Omron Sysmac Studio project Auto Connect Project (Sysmac Studio 1.48.0.8, StandardProject)

# Controller new_Controller_0: NX102-1020 version 1.35
Units and slaves: Unit 1 : NX-CIF101 (N1); Unit 2 : NX-ID5142-1 (N2); Unit 3 : NX-OD5121-1 (N3)
Task PrimaryTask (priority 4, period or condition 2000): Program0

VAR_GLOBAL RETAIN
    data1 : INT;
END_VAR
VAR_GLOBAL
    data2 : INT;
    data3 : INT;
    data4 : INT;
    data5 : INT;
    dataA_1 : STRING[256];
    dataA_2 : STRING[256];
    dataA_3 : STRING[256];
    dataA_4 : STRING[256];
    dataA_5 : STRING[256];
    dataB_1 : REAL;
    dataB_2 : REAL;
    dataB_3 : REAL;
    dataB_4 : REAL;
    dataB_5 : REAL;
    senser1 : BOOL;
    pump1 : BOOL;
    pb_start : BOOL;
END_VAR

PROGRAM Program0
VAR
    start_1 : BOOL;
    stop_1 : BOOL;
    lam_1 : BOOL;
    lamp_1 : BOOL;
    sw_1 : BOOL;
    sw2 : BOOL;
    sw_2 : BOOL;
    lamp_2 : BOOL;
    sw3 : BOOL;
    sw4 : BOOL;
    lamp_3 : BOOL;
    sw5 : BOOL;
    lamp_4 : BOOL;
    sw_6 : BOOL;
    lamp_5 : BOOL;
    sw7 : BOOL;
    test_a : RS;
    sw_test_a : BOOL;
    lamp_6 : BOOL;
    sw_9 : BOOL;
    sww : BOOL;
    sw_8 : BOOL;
    test_b : BOOL;
    lamp_7 : BOOL;
    test_a_q1 : BOOL;
    sw_10 : BOOL;
    lamp_8 : BOOL;
    sw_11 : BOOL;
    test_b_1 : SR;
    t_on : BOOL;
    t_a1 : TON;
    pv1 : TIME;
    lamp_9 : BOOL;
    t_b1 : TOF;
    sw12 : BOOL;
    pv2 : TIME;
    lamp_10 : BOOL;
    sw13 : BOOL;
    t_c1 : TP;
    pv3 : TIME;
    lamp_11 : BOOL;
    sw14 : BOOL;
    t_d1 : AccumulationTimer;
    sw15 : BOOL;
    pv4 : TIME;
    lamp_12 : BOOL;
    C_A_D_C : CTU;
    box2 : BOOL;
    box1 : BOOL;
    pd_reset_1 : BOOL;
    cv_1 : INT;
    lamp_13 : BOOL;
    sw16 : BOOL;
    sw_17 : BOOL;
    sw_18 : BOOL;
    lamp_test : BOOL;
    sw_19 : BOOL;
    lamp_14 : BOOL;
    B1 : BOOL;
    B2 : BOOL;
    B3 : BOOL;
    B4 : BOOL;
    B5 : BOOL;
    B6 : BOOL;
    B7 : BOOL;
    lamp_15 : BOOL;
    p : BOOL;
END_VAR
VAR_EXTERNAL
    data1 : INT;
    data2 : INT;
    dataA_1 : STRING[256];
    dataA_2 : STRING[256];
    data3 : INT;
    data4 : INT;
    dataB_1 : REAL;
    dataB_2 : REAL;
    senser1 : BOOL;
    pump1 : BOOL;
END_VAR
VAR
    _t1 : BOOL;
    _e2 : F_TRIG;
    _e3 : R_TRIG;
    _e4 : R_TRIG;
END_VAR

(* Section Section0: ladder, written here as Structured Text *)

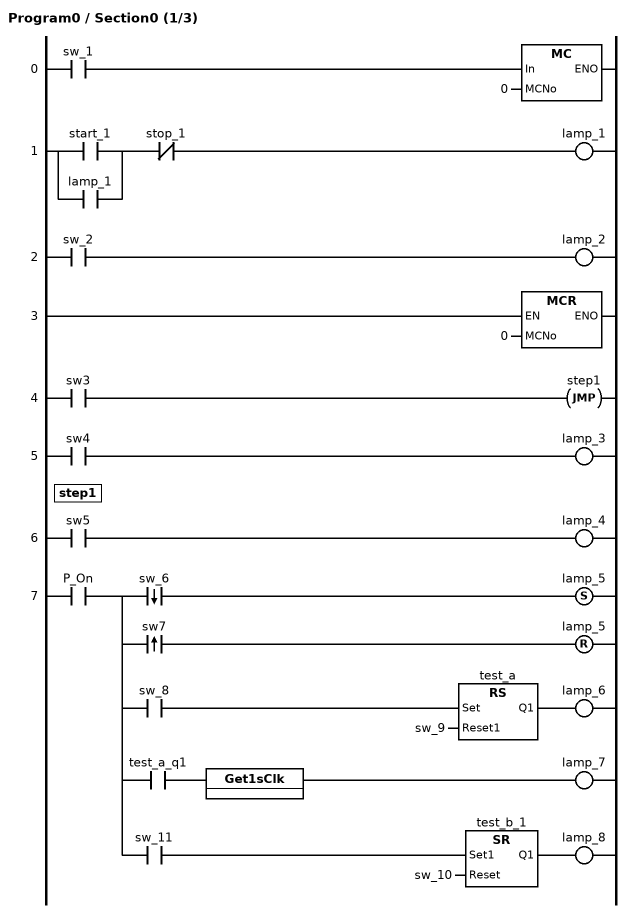
(* Rung 0 *)
MC(In := sw_1, MCNo := 0, ENO => _t1);
(* Rung 1 *)
lamp_1 := (start_1 OR lamp_1) AND NOT stop_1;
(* Rung 2 *)
lamp_2 := sw_2;
(* Rung 3 *)
MCR(MCNo := 0);
(* Rung 4 *)
IF sw3 THEN JMP step1; END_IF;
(* Rung 5 *)
lamp_3 := sw4;
(* Rung 6 *)
step1:
lamp_4 := sw5;
(* Rung 7 *)
_e2(CLK := sw_6);
IF P_On AND _e2.Q THEN lamp_5 := TRUE; END_IF;
_e3(CLK := sw7);
IF P_On AND _e3.Q THEN lamp_5 := FALSE; END_IF;
test_a(Set := P_On AND sw_8, Reset1 := sw_9);
lamp_6 := test_a.Q1;
lamp_7 := P_On AND test_a_q1 AND Get1sClk();
test_b_1(Set1 := P_On AND sw_11, Reset := sw_10);
lamp_8 := test_b_1.Q1;

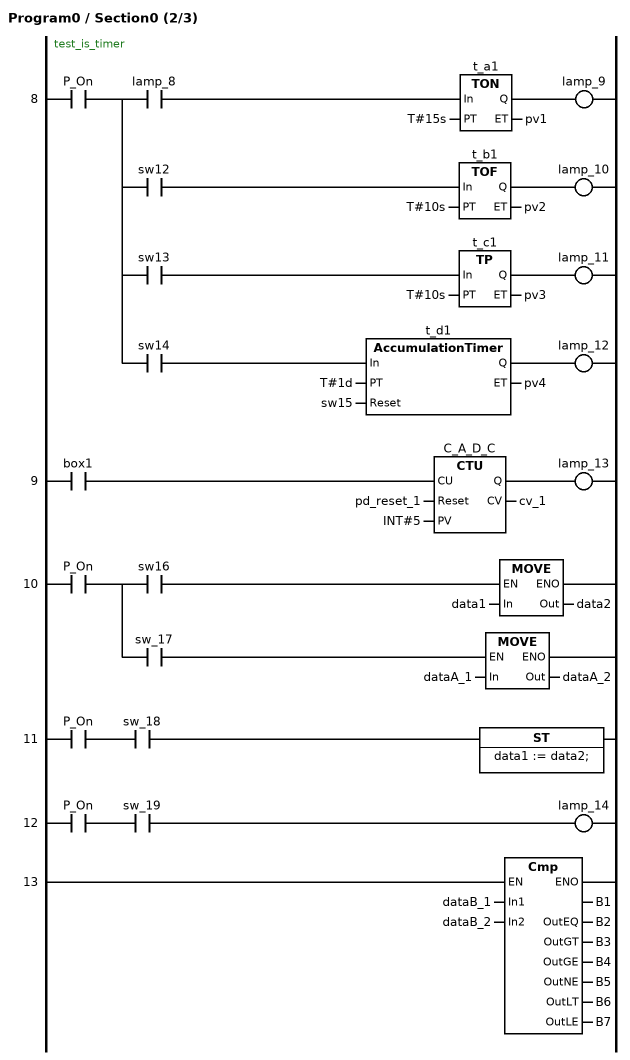
(* Rung 8: test_is_timer *)
t_a1(In := P_On AND lamp_8, PT := T#15s, ET => pv1);
lamp_9 := t_a1.Q;
t_b1(In := P_On AND sw12, PT := T#10s, ET => pv2);
lamp_10 := t_b1.Q;
t_c1(In := P_On AND sw13, PT := T#10s, ET => pv3);
lamp_11 := t_c1.Q;
t_d1(In := P_On AND sw14, PT := T#1d, Reset := sw15, ET => pv4);
lamp_12 := t_d1.Q;
(* Rung 9 *)
_e4(CLK := box1);
C_A_D_C(CU := _e4.Q, Reset := pd_reset_1, PV := INT#5, CV => cv_1);
lamp_13 := C_A_D_C.Q;
(* Rung 10 *)
IF P_On AND sw16 THEN data2 := data1; END_IF;
IF P_On AND sw_17 THEN dataA_2 := dataA_1; END_IF;
(* Rung 11 *)
IF P_On AND sw_18 THEN
    data1 := data2;
END_IF;
(* Rung 12 *)
lamp_14 := P_On AND sw_19;
(* Rung 13 *)
B1 := Cmp(In1 := dataB_1, In2 := dataB_2, OutEQ => B2, OutGT => B3, OutGE => B4, OutNE => B5, OutLT => B6, OutLE => B7);

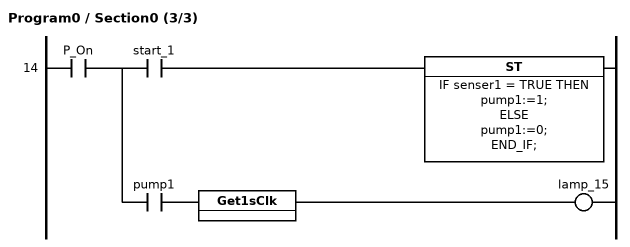
(* Rung 14 *)
IF P_On AND start_1 THEN
    IF senser1 = TRUE THEN
    	pump1:=1;
    ELSE
    	pump1:=0;
    END_IF;
END_IF;
lamp_15 := P_On AND pump1 AND Get1sClk();
END_PROGRAM